// TwinCAT 3 PLC project Untitled1
// ProgramVersion: 3.1.4024.0
// libraries:
//   JSC_MC_Lib, * (Jenny Science AG)
//   JS_MC_REF, * (Jenny Science AG)
//   Tc2_MC2, * (Beckhoff Automation GmbH)
//   Tc2_NC, * (Beckhoff Automation GmbH)
//   Tc2_Standard, * (Beckhoff Automation GmbH)
//   Tc2_System, * (Beckhoff Automation GmbH)
//   Tc2_Utilities, * (Beckhoff Automation GmbH)
//   Tc3_Module, * (Beckhoff Automation GmbH)
//   BASIC,3.3.3.0,OSCAT
// project tree:
//   / PlcTask.TcTTO
//   POUs/ FB_Button.TcPOU, FB_LongPress.TcPOU, FB_XAxis.TcPOU, FB_Yaxis.TcPOU, MAIN.TcPOU
// real-time tasks:
//   TASK PlcTask: cycle T#10ms, priority 20, ADS port 350
// I/O:
//   DEVICE Device 2 (EtherCAT), AmsNetId 10.0.3.17.3.1
//     Drive 1 (Xvi) [XENAX Xvi 48V8]
//     Drive 2 (Xvi) [XENAX Xvi 48V8]
//     Box 3 (EPP2334-0061) [EPP2334-0061 4 Ch. Dig. Input/Output 24V, 0,5A, M8]
//     Box 4 (EPP9001-0060) [EPP9001-0060 4 K. Dig. EtherCAT P / EtherCAT ECP/EC Connector with voltage forwarding]
// variable links:
//   Untitled1/Untitled1 Instance <-> Device 2 (EtherCAT)/Box 3 (EPP2334-0061)
//     PlcTask Inputs/MAIN.FB_Button.ButtonInput <-> Channel 1/Input
//     PlcTask Inputs/MAIN.FB_LongPress.Button <-> Channel 1/Input
//     PlcTask Outputs/MAIN.FB_Button.ButtonLight <-> Channel 6/Output
//   Untitled1/Untitled1 Instance <-> Device 2 (EtherCAT)/Drive 1 (Xvi)
//     PlcTask Inputs/MAIN.Xaxis.instJS_MC_Init.RxPDO/bWcState <-> WcState/WcState
//     PlcTask Inputs/MAIN.Xaxis.instJS_MC_Init.RxPDO/diPositionActualValue_I6064 <-> TxPDO 5/Position Actual Value
//     PlcTask Inputs/MAIN.Xaxis.instJS_MC_Init.RxPDO/diProcessStatusRegister_I2006 <-> TxPDO 5/Process Status Register
//     PlcTask Inputs/MAIN.Xaxis.instJS_MC_Init.RxPDO/uiStatusword_I6041 <-> TxPDO 5/Statusword
//     PlcTask Inputs/MAIN.Xaxis.instJS_MC_Init.stSlaveAmsAddr/netId <-> InfoData/AdsAddr/netId
//     PlcTask Inputs/MAIN.Xaxis.instJS_MC_Init.stSlaveAmsAddr/port <-> InfoData/AdsAddr/port
//     PlcTask Outputs/MAIN.Xaxis.instJS_MC_Init.TxPDO/diTargetPosition_I607A <-> RxPDO 5/Target Position
//     PlcTask Outputs/MAIN.Xaxis.instJS_MC_Init.TxPDO/udiProfileAcceleration_I6083 <-> RxPDO 5/Profile Acceleration
//     PlcTask Outputs/MAIN.Xaxis.instJS_MC_Init.TxPDO/udiProfileVelocity_I6081 <-> RxPDO 5/Profile Velocity
//     PlcTask Outputs/MAIN.Xaxis.instJS_MC_Init.TxPDO/udiS_CurveProfile_I2000 <-> RxPDO 5/S-Curve Profile
//     PlcTask Outputs/MAIN.Xaxis.instJS_MC_Init.TxPDO/uiControlword_I6040 <-> RxPDO 5/Controlword
//   Untitled1/Untitled1 Instance <-> Device 2 (EtherCAT)/Drive 2 (Xvi)
//     PlcTask Inputs/MAIN.Yaxis.instJS_MC_Init.RxPDO/bWcState <-> WcState/WcState
//     PlcTask Inputs/MAIN.Yaxis.instJS_MC_Init.RxPDO/diPositionActualValue_I6064 <-> TxPDO 5/Position Actual Value
//     PlcTask Inputs/MAIN.Yaxis.instJS_MC_Init.RxPDO/diProcessStatusRegister_I2006 <-> TxPDO 5/Process Status Register
//     PlcTask Inputs/MAIN.Yaxis.instJS_MC_Init.RxPDO/uiStatusword_I6041 <-> TxPDO 5/Statusword
//     PlcTask Inputs/MAIN.Yaxis.instJS_MC_Init.stSlaveAmsAddr/netId <-> InfoData/AdsAddr/netId
//     PlcTask Inputs/MAIN.Yaxis.instJS_MC_Init.stSlaveAmsAddr/port <-> InfoData/AdsAddr/port
//     PlcTask Outputs/MAIN.Yaxis.instJS_MC_Init.TxPDO/diTargetPosition_I607A <-> RxPDO 5/Target Position
//     PlcTask Outputs/MAIN.Yaxis.instJS_MC_Init.TxPDO/udiProfileAcceleration_I6083 <-> RxPDO 5/Profile Acceleration
//     PlcTask Outputs/MAIN.Yaxis.instJS_MC_Init.TxPDO/udiProfileVelocity_I6081 <-> RxPDO 5/Profile Velocity
//     PlcTask Outputs/MAIN.Yaxis.instJS_MC_Init.TxPDO/udiS_CurveProfile_I2000 <-> RxPDO 5/S-Curve Profile
//     PlcTask Outputs/MAIN.Yaxis.instJS_MC_Init.TxPDO/uiControlword_I6040 <-> RxPDO 5/Controlword

CONFIGURATION Untitled1
    RESOURCE PLC ON TwinCAT3
        TASK PlcTask(INTERVAL := T#10ms, PRIORITY := 20);
        PROGRAM MAIN WITH PlcTask : MAIN;
    END_RESOURCE
END_CONFIGURATION

// ---- POUs/MAIN.TcPOU
PROGRAM MAIN
VAR
	nPosition : DINT := 60000;
	Yaxis : FB_XAxis;
	Xaxis : FB_Yaxis;
	bBool : BOOL := FALSE;
	FB_Button : FB_Button;
	FB_LongPress : FB_LongPress;
	FB_Reset : TC_RESTART;
END_VAR

Yaxis(bMotorOn := FB_Button.bMotorOn);
Xaxis(bToken := Yaxis.bYstart, FlipProcess := FB_Button.FlipProcess);
FB_Button(ProcessFinished := Xaxis.bProcessFinished);
FB_LongPress();
FB_Reset(RESTART := FB_LongPress.bReset);

END_PROGRAM

// ---- POUs/FB_XAxis.TcPOU
FUNCTION_BLOCK PUBLIC FB_XAxis
VAR_INPUT
	bMotorOn : BOOL;
END_VAR

VAR
	fbTon : TON := (PT :=T#1.5S);
	nMoveCount : DINT := 0;
	Enable_Prog_Functions : BOOL := TRUE; (* Start demo *)
    state : INT; (*-10: connection lost, -20/-21: Error, 100-199 demo application, 200: idle state*)
    
	CommunicationError : BOOL; (* No Communication to XENAX*)	
    ValidConCnt : INT; (*CyclicIn.valid toggles somtetimes. So we believe the CyclicIn.valid only after some time*)
	
	  (*Function blocks required for operation*)
  instJS_MC_Init 					: JS_MC_Init;
  instJS_MC_CyclicIn 				: JS_MC_CyclicIn;
  instJS_MC_CyclicOut 			: JS_MC_CyclicOut;
  instJS_MC_Power 				: JS_MC_Power;
  instJS_MC_Reference 			: JS_MC_Reference;
  instJS_MC_Stop 					: JS_MC_Stop;
  instJS_MC_Reset 				: JS_MC_Reset;
  
  (*Additional function blocks for Profile Position*)
  	instJS_MC_MoveAbsolute 			: JS_MC_MoveAbsolute;
  	instJS_MC_MoveRelative 			: JS_MC_MoveRelative;
  	instJS_MC_JogVelocity			: JS_MC_JogVelocity;
  	instJS_MC_Halt 					: JS_MC_Halt;
	
  (*Function blocks for error handling*)
  	instJS_MC_ReadAxisError			: JS_MC_ReadAxisError;
  	instJS_MC_AxisErrorCollector	: JS_MC_AxisErrorCollector;
	
  (*Optional function blocks*)
	instJS_MC_ReadActualPosition 	: JS_MC_ReadActualPosition;
	instJS_MC_ReadStatus 			: JS_MC_ReadStatus;
	instJS_MC_ReadPSR	 			: JS_MC_ReadPSR;
	instJS_MC_ReadDigitalOutput 	: JS_MC_ReadDigitalOutput;
	instJS_MC_ReadDigitalInput 		: JS_MC_ReadDigitalInput;
	instJS_MC_ReadParameter 		: JS_MC_ReadParameter;
	instJS_MC_WriteParameter 		: JS_MC_WriteParameter;
	instJS_MC_WriteDigitalOutput 	: JS_MC_WriteDigitalOutput;
END_VAR

VAR_OUTPUT 
	bYstart : BOOL;
END_VAR

IF NOT instJS_MC_Init.Valid THEN
    instJS_MC_Init.OperationMode := gcJS_MC.jsmcMODE_PROFILE_POSITION; //PROFILE_POSITION: trajectories are calculated by Xenax Servocontroller. There is no need for an NC Axis, less PLC cpu consumption, but gives less control over driving behavior.
    instJS_MC_Init();                         // init Axis, only call this funtion once at startup
    
    (*reference options*)
    instJS_MC_Reference.ReferenceMode	:= gcJS_MC.jsmcREFERENCE_MODE_DEFAULT;      (* Motor type specific default reference method*)
    (*additional reference options for rotative motors*)
    instJS_MC_Reference.ZMarkSpeedRot := 10000;                                   (* speed during refernce*)
    instJS_MC_Reference.ReferenceSpeedRot := 0;                                   (* speed for optional refernce to a home sensor, 0 is disabled*)
    
    (*enable Error and Status block*)
    instJS_MC_ReadAxisError.Enable := TRUE;
    instJS_MC_ReadStatus.Enable := TRUE;

(***********************************************************************************
 * run loop
 ***********************************************************************************)
ELSE
    instJS_MC_Init(); //recall JS_MC_Init is required for online changes. It recalculates pstAxis output.
    instJS_MC_CyclicIn(pstAxis := instJS_MC_Init.pstAxis); //Gets cyclic data from EtherCat bus und checks if connection is still valid

	IF instJS_MC_CyclicIn.Error AND state >= 0 THEN (*handle Communication Error e.g. ethernet cable disconnected if not already on error*)
        state := -10;
	END_IF
(*-------------------------------------------------------------------------------------------------------------------------------*)

    CASE state OF 
    (*Power Up sequence----------------------------------------------------------------------------------------------------------*)
	0:	(*enable instJS_MC_CyclicIn*)
        IF Enable_Prog_Functions THEN
            instJS_MC_CyclicIn.Enable := TRUE;
            ValidConCnt := 0;
            state := 1;
        END_IF;
        
    1:  (*wait instJS_MC_CyclicIn valid is stable*)
        IF instJS_MC_CyclicIn.Valid THEN
            ValidConCnt := ValidConCnt + 1;
            IF ValidConCnt >= 15 THEN
                CommunicationError := FALSE;
                state := 2;
			END_IF
		END_IF
        
    2:  (* reset erros from previous run*)
		instJS_MC_Reset.Execute := TRUE;
		state := 3;        
	
	3:  
    	IF instJS_MC_Reset.Done THEN
			instJS_MC_Reset.Execute := FALSE;
			state := 10;
		END_IF
							
	10: (* power on*)
		instJS_MC_Power.Enable := 1;
        state := 11;
        
    11:
		IF instJS_MC_Power.Status AND instJS_MC_Power.Valid THEN
            state := 30;
		END_IF

	30: (* start reference*)
		instJS_MC_Reference.Execute := TRUE;
		state := 31;
	
	31:
		IF instJS_MC_Reference.Done THEN
			instJS_MC_Reference.Execute := FALSE;
			state := 100;
		END_IF
    (*normal operation of demo application-------------------------------------------------------------------------------------------------------------*)
	100: (*drive to position 0*)
		instJS_MC_MoveAbsolute.Execute := TRUE;
		instJS_MC_MoveAbsolute.Position := 0;           //increment
		nMoveCount := 10000;
		instJS_MC_MoveAbsolute.Velocity := 100000;       //increment/s
		instJS_MC_MoveAbsolute.Acceleration := 1000000; //increment/s^2
		instJS_MC_MoveAbsolute.Scurve := 50;            //"smoothness" or change of acceleration in %
		state := 101;
		bYstart := FALSE;
	
	101:
		IF instJS_MC_MoveAbsolute.Done THEN
			instJS_MC_MoveAbsolute.Execute := FALSE;
			state := 102;
 		END_IF

	102: (*drive to position 40000*)
		IF bMotorOn THEN
			instJS_MC_MoveAbsolute.Execute := TRUE;
			instJS_MC_MoveAbsolute.Position := nMoveCount;       //increment
			nMoveCount := nMoveCount + 5000;
			instJS_MC_MoveAbsolute.Velocity := 50000;       //increment/s
			instJS_MC_MoveAbsolute.Acceleration := 1000000; //increment/s^2
			instJS_MC_MoveAbsolute.Scurve := 50;            //"smoothness" or change of acceleration in %
			state := 103;
		END_IF
	
	103:
	fbTon(IN := TRUE);
	IF fbTON.Q THEN
		fbTON(IN := FALSE);
		IF instJS_MC_MoveAbsolute.Done THEN
			instJS_MC_MoveAbsolute.Execute := FALSE;
            IF Enable_Prog_Functions THEN
				IF nMoveCount >= 75000 THEN 
					bYstart := TRUE;
					state := 100;
				ELSE
                	state := 101;   //restart
            	END_IF    
 			END_IF
    	END_IF
	END_IF
	
    200:(*idle state*)
        IF Enable_Prog_Functions THEN
            state := 100;
        END_IF    

    (*error handling-----------------------------------------------------------------------------------------------------------------------*)
    -10: (* Communication interrupted, reset variables and try to reconnect*)
        CommunicationError := TRUE;
		instJS_MC_CyclicIn.Enable := FALSE;
        
        instJS_MC_Reset.Execute := FALSE;
		instJS_MC_Reference.Execute := FALSE;
		instJS_MC_Power.Enable := FALSE;
		instJS_MC_MoveAbsolute.Execute := FALSE;
        state := 0;
        
    -20: (*Axis error during normal operation*)
        instJS_MC_Reset.Execute := FALSE;
		instJS_MC_Reference.Execute := FALSE;
		instJS_MC_Power.Enable := FALSE;
		instJS_MC_MoveAbsolute.Execute := FALSE;
        state := -21;
        
    -21:
        //instJS_MC_Reset.Execute := true; (*acknowledge axis error over hmi for example*)


    END_CASE

	(* Call all JS_MC_Lib function blocks if CyclicIn is Valid-------------------------------------------------------------------------------*)
    IF instJS_MC_CyclicIn.Valid THEN
        (*Function blocks required for operation*)
        instJS_MC_Power( pstAxis := instJS_MC_Init.pstAxis);
        instJS_MC_Reference( pstAxis := instJS_MC_Init.pstAxis);
        instJS_MC_Stop( pstAxis := instJS_MC_Init.pstAxis);
        instJS_MC_Reset( pstAxis := instJS_MC_Init.pstAxis);
        (*Additional function blocks for Profile Position*)
        instJS_MC_MoveAbsolute( pstAxis := instJS_MC_Init.pstAxis);
        instJS_MC_MoveRelative( pstAxis := instJS_MC_Init.pstAxis);
        instJS_MC_JogVelocity( pstAxis := instJS_MC_Init.pstAxis);
        instJS_MC_Halt( pstAxis := instJS_MC_Init.pstAxis);
        (*Function blocks for error handling*)
        instJS_MC_ReadAxisError( pstAxis := instJS_MC_Init.pstAxis);
        instJS_MC_AxisErrorCollector( pstAxis := instJS_MC_Init.pstAxis);
        (*Optional function blocks*)
        instJS_MC_ReadActualPosition( pstAxis := instJS_MC_Init.pstAxis);
        instJS_MC_ReadStatus( pstAxis := instJS_MC_Init.pstAxis);
        instJS_MC_ReadPSR( pstAxis := instJS_MC_Init.pstAxis);
        instJS_MC_ReadDigitalOutput( pstAxis := instJS_MC_Init.pstAxis);
        instJS_MC_ReadDigitalInput( pstAxis := instJS_MC_Init.pstAxis);
        instJS_MC_ReadParameter( pstAxis := instJS_MC_Init.pstAxis);
        instJS_MC_WriteParameter( pstAxis := instJS_MC_Init.pstAxis);
        instJS_MC_WriteDigitalOutput( pstAxis := instJS_MC_Init.pstAxis);
    END_IF
    //always call cyclic out
	instJS_MC_CyclicOut( pstAxis := instJS_MC_Init.pstAxis);
END_IF

END_FUNCTION_BLOCK

// ---- POUs/FB_Yaxis.TcPOU
FUNCTION_BLOCK PUBLIC FB_Yaxis
VAR_INPUT
	bToken : BOOL;
	FlipProcess : BOOL; 
END_VAR

VAR
	nMoveCount : DINT := 60000; //Position of Linear Motor
	fbTon : TON := (PT :=T#5S); // Timer for scanning in QR 
	Enable_Prog_Functions : BOOL := TRUE; (* Start demo *)
    state : INT; (*-10: connection lost, -20/-21: Error, 100-199 demo application, 200: idle state*)
    
	CommunicationError : BOOL; (* No Communication to XENAX*)	
    ValidConCnt : INT; (*CyclicIn.valid toggles somtetimes. So we believe the CyclicIn.valid only after some time*)
	
	  (*Function blocks required for operation*)
  instJS_MC_Init 					: JS_MC_Init;
  instJS_MC_CyclicIn 				: JS_MC_CyclicIn;
  instJS_MC_CyclicOut 			: JS_MC_CyclicOut;
  instJS_MC_Power 				: JS_MC_Power;
  instJS_MC_Reference 			: JS_MC_Reference;
  instJS_MC_Stop 					: JS_MC_Stop;
  instJS_MC_Reset 				: JS_MC_Reset;
  
  (*Additional function blocks for Profile Position*)
  	instJS_MC_MoveAbsolute 			: JS_MC_MoveAbsolute;
  	instJS_MC_MoveRelative 			: JS_MC_MoveRelative;
  	instJS_MC_JogVelocity			: JS_MC_JogVelocity;
  	instJS_MC_Halt 					: JS_MC_Halt;
	
  (*Function blocks for error handling*)
  	instJS_MC_ReadAxisError			: JS_MC_ReadAxisError;
  	instJS_MC_AxisErrorCollector	: JS_MC_AxisErrorCollector;
	
  (*Optional function blocks*)
	instJS_MC_ReadActualPosition 	: JS_MC_ReadActualPosition;
	instJS_MC_ReadStatus 			: JS_MC_ReadStatus;
	instJS_MC_ReadPSR	 			: JS_MC_ReadPSR;
	instJS_MC_ReadDigitalOutput 	: JS_MC_ReadDigitalOutput;
	instJS_MC_ReadDigitalInput 		: JS_MC_ReadDigitalInput;
	instJS_MC_ReadParameter 		: JS_MC_ReadParameter;
	instJS_MC_WriteParameter 		: JS_MC_WriteParameter;
	instJS_MC_WriteDigitalOutput 	: JS_MC_WriteDigitalOutput;
END_VAR

VAR_OUTPUT 
	bProcessFinished : BOOL; 
END_VAR

IF NOT instJS_MC_Init.Valid THEN
    instJS_MC_Init.OperationMode := gcJS_MC.jsmcMODE_PROFILE_POSITION; //PROFILE_POSITION: trajectories are calculated by Xenax Servocontroller. There is no need for an NC Axis, less PLC cpu consumption, but gives less control over driving behavior.
    instJS_MC_Init();                         // init Axis, only call this funtion once at startup
    
    (*reference options*)
    instJS_MC_Reference.ReferenceMode	:= gcJS_MC.jsmcREFERENCE_MODE_DEFAULT;      (* Motor type specific default reference method*)
    (*additional reference options for rotative motors*)
    instJS_MC_Reference.ZMarkSpeedRot := 10000;                                   (* speed during refernce*)
    instJS_MC_Reference.ReferenceSpeedRot := 0;                                   (* speed for optional refernce to a home sensor, 0 is disabled*)
    
    (*enable Error and Status block*)
    instJS_MC_ReadAxisError.Enable := TRUE;
    instJS_MC_ReadStatus.Enable := TRUE;

(***********************************************************************************
 * run loop
 ***********************************************************************************)
ELSE
    instJS_MC_Init(); //recall JS_MC_Init is required for online changes. It recalculates pstAxis output.
    instJS_MC_CyclicIn(pstAxis := instJS_MC_Init.pstAxis); //Gets cyclic data from EtherCat bus und checks if connection is still valid

	IF instJS_MC_CyclicIn.Error AND state >= 0 THEN (*handle Communication Error e.g. ethernet cable disconnected if not already on error*)
        state := -10;
	END_IF
(*-------------------------------------------------------------------------------------------------------------------------------*)

    CASE state OF 
    (*Power Up sequence----------------------------------------------------------------------------------------------------------*)
	0:	(*enable instJS_MC_CyclicIn*)
        IF Enable_Prog_Functions THEN
            instJS_MC_CyclicIn.Enable := TRUE;
            ValidConCnt := 0;
            state := 1;
        END_IF;
        
    1:  (*wait instJS_MC_CyclicIn valid is stable*)
        IF instJS_MC_CyclicIn.Valid THEN
            ValidConCnt := ValidConCnt + 1;
            IF ValidConCnt >= 15 THEN
                CommunicationError := FALSE;
                state := 2;
			END_IF
		END_IF
        
    2:  (* reset erros from previous run*)
		instJS_MC_Reset.Execute := TRUE;
		state := 3;        
	
	3:  
    	IF instJS_MC_Reset.Done THEN
			instJS_MC_Reset.Execute := FALSE;
			state := 10;
		END_IF
							
	10: (* power on*)
		instJS_MC_Power.Enable := 1;
        state := 11;
        
    11:
		IF instJS_MC_Power.Status AND instJS_MC_Power.Valid THEN
            state := 30;
		END_IF

	30: (* start reference*)
		instJS_MC_Reference.Execute := TRUE;
		state := 31;
	
	31:
		IF instJS_MC_Reference.Done THEN
			instJS_MC_Reference.Execute := FALSE;
			state := 100;
		END_IF
    (*normal operation of demo application-------------------------------------------------------------------------------------------------------------*)
	100: (*drive to position 0*)
		IF nMoveCount < 0 THEN
			nMoveCount := 60000;
			bProcessFinished := TRUE;
		END_IF
		instJS_MC_MoveAbsolute.Execute := TRUE;
		instJS_MC_MoveAbsolute.Position := nMoveCount;           //increment
		nMoveCount := nMoveCount - 20000;
		instJS_MC_MoveAbsolute.Velocity := 100000;       //increment/s
		instJS_MC_MoveAbsolute.Acceleration := 1000000; //increment/s^2
		instJS_MC_MoveAbsolute.Scurve := 50;            //"smoothness" or change of acceleration in %
		state := 101;
	
	101:
	fbTon(IN := TRUE);
	IF fbTON.Q THEN
		fbTON(IN := FALSE);
		IF instJS_MC_MoveAbsolute.Done THEN
			instJS_MC_MoveAbsolute.Execute := FALSE;
			state := 103;
 		END_IF
	END_IF
	
	103:
	bProcessFinished := FlipProcess;
	IF bToken THEN
		IF instJS_MC_MoveAbsolute.Done THEN
			instJS_MC_MoveAbsolute.Execute := FALSE;
            IF Enable_Prog_Functions THEN
                	state := 100;   //restart
 			END_IF
    	END_IF
		bToken := FALSE;
	END_IF
	
    200:(*idle state*)
        IF Enable_Prog_Functions THEN
            state := 100;
        END_IF    

    (*error handling-----------------------------------------------------------------------------------------------------------------------*)
    -10: (* Communication interrupted, reset variables and try to reconnect*)
        CommunicationError := TRUE;
		instJS_MC_CyclicIn.Enable := FALSE;
        
        instJS_MC_Reset.Execute := FALSE;
		instJS_MC_Reference.Execute := FALSE;
		instJS_MC_Power.Enable := FALSE;
		instJS_MC_MoveAbsolute.Execute := FALSE;
        state := 0;
        
    -20: (*Axis error during normal operation*)
        instJS_MC_Reset.Execute := FALSE;
		instJS_MC_Reference.Execute := FALSE;
		instJS_MC_Power.Enable := FALSE;
		instJS_MC_MoveAbsolute.Execute := FALSE;

    END_CASE

	(* Call all JS_MC_Lib function blocks if CyclicIn is Valid-------------------------------------------------------------------------------*)
    IF instJS_MC_CyclicIn.Valid THEN
        (*Function blocks required for operation*)
        instJS_MC_Power( pstAxis := instJS_MC_Init.pstAxis);
        instJS_MC_Reference( pstAxis := instJS_MC_Init.pstAxis);
        instJS_MC_Stop( pstAxis := instJS_MC_Init.pstAxis);
        instJS_MC_Reset( pstAxis := instJS_MC_Init.pstAxis);
        (*Additional function blocks for Profile Position*)
        instJS_MC_MoveAbsolute( pstAxis := instJS_MC_Init.pstAxis);
        instJS_MC_MoveRelative( pstAxis := instJS_MC_Init.pstAxis);
        instJS_MC_JogVelocity( pstAxis := instJS_MC_Init.pstAxis);
        instJS_MC_Halt( pstAxis := instJS_MC_Init.pstAxis);
        (*Function blocks for error handling*)
        instJS_MC_ReadAxisError( pstAxis := instJS_MC_Init.pstAxis);
        instJS_MC_AxisErrorCollector( pstAxis := instJS_MC_Init.pstAxis);
        (*Optional function blocks*)
        instJS_MC_ReadActualPosition( pstAxis := instJS_MC_Init.pstAxis);
        instJS_MC_ReadStatus( pstAxis := instJS_MC_Init.pstAxis);
        instJS_MC_ReadPSR( pstAxis := instJS_MC_Init.pstAxis);
        instJS_MC_ReadDigitalOutput( pstAxis := instJS_MC_Init.pstAxis);
        instJS_MC_ReadDigitalInput( pstAxis := instJS_MC_Init.pstAxis);
        instJS_MC_ReadParameter( pstAxis := instJS_MC_Init.pstAxis);
        instJS_MC_WriteParameter( pstAxis := instJS_MC_Init.pstAxis);
        instJS_MC_WriteDigitalOutput( pstAxis := instJS_MC_Init.pstAxis);
    END_IF
    //always call cyclic out
	instJS_MC_CyclicOut( pstAxis := instJS_MC_Init.pstAxis);
END_IF

END_FUNCTION_BLOCK

// ---- POUs/FB_Button.TcPOU
FUNCTION_BLOCK PUBLIC FB_Button
VAR_INPUT
	ProcessFinished : BOOL;
END_VAR

VAR
	ButtonInput AT%I* : BOOL;
	ButtonLight AT%Q* : BOOL := TRUE;
	Click : F_TRIG;
	fbTon : TON := (PT :=T#0.3S); 
	state : INT := 0;
END_VAR

VAR_OUTPUT
	bMotorOn : BOOL;
	FlipProcess : BOOL; 
END_VAR

CASE state OF
	
	0:
		Click(CLK := ButtonInput);
		IF Click.Q THEN
			state := 20;
			FlipProcess := FALSE;
		END_IF
		fbTon(IN := TRUE);
		IF fbTON.Q THEN
			fbTON(IN := FALSE);	
			ButtonLight := FALSE;
			state := 10;
		END_IF
		bMotorOn := FALSE;
		
	10:
		Click(CLK := ButtonInput);
		IF Click.Q THEN
			state := 20;
			FlipProcess := FALSE;
		END_IF
		fbTon(IN := TRUE);
		IF fbTON.Q THEN
			fbTON(IN := FALSE);	
			ButtonLight := TRUE;
			state := 0;
		END_IF
		bMotorOn := FALSE;
		
	20: 
		Click(CLK := ButtonInput);
		IF Click.Q  OR ProcessFinished THEN
			state := 0;
		END_IF
		ButtonLight := TRUE;	
		bMotorOn := TRUE;
	
END_CASE

END_FUNCTION_BLOCK

// ---- POUs/FB_LongPress.TcPOU
FUNCTION_BLOCK FB_LongPress
VAR_OUTPUT
	bReset : BOOL;
END_VAR

VAR
	state : INT := 0;
	Button AT%I* : BOOL;
	fbTon : TON := (PT :=T#3S); 
END_VAR

CASE state OF
	0:
		fbTon(IN := FALSE);
		IF Button THEN 
			state := 10;
		END_IF
		
	10:
		fbTon(IN := TRUE);
		IF fbTon.Q THEN 
			IF Button THEN
				bReset := TRUE;
			END_IF
			state := 0;
		END_IF
		IF NOT BUTTON THEN 
			state := 0;
		END_IF
		
END_CASE

END_FUNCTION_BLOCK
